Fanuc KAREL source: NC0015.KL

-- PROVISIONAL review KL for V940-1; original PC SHA256 a06a1c527e8287789b05f7df9faa5f540ba820ada4ca568a80dea30cb171e11d
-- Incomplete behavior may be omitted. Consult companion uncertainty JSON. Do not deploy.
PROGRAM NC0015
%NOLOCKGROUP
-- UNRESOLVED_LOCAL_POOL 1 cells at code offset 3; source declarations unknown
-- DIRECT_LOCAL_WORD_ACCESS alone does not prove INTEGER, REAL, or BOOLEAN
BEGIN
  -- V9_EXPOSED_INDEXED_TABLE_HINT layout=0001; 10 counted words exposed once; source arms/runtime held
  -- V9_CONDITION_STACK_HINT 5 bounded expression windows; static native code-base-relative target link; source arms held
  -- UNRESOLVED_PC offsets 0-8; opcodes 2B,2C,7B
  -- UNRESOLVED_PC offsets 13-20; opcodes 9D,23
  -- UNRESOLVED_PC offsets 25-38; opcodes 21,9D,57,79
  -- UNRESOLVED_PC offsets 43-61; opcodes 21,2E,52,23
  -- UNRESOLVED_PC offsets 66-71; opcodes 7A
  -- UNRESOLVED_PC offsets 76-89; opcodes 21,9D,57,79
  -- UNRESOLVED_PC offsets 94-112; opcodes 21,2E,52,23
  -- UNRESOLVED_PC offsets 117-122; opcodes 7A
  -- UNRESOLVED_PC offsets 127-140; opcodes 21,9D,57,79
  -- UNRESOLVED_PC offsets 145-163; opcodes 21,2E,52,23
  -- UNRESOLVED_PC offsets 168-173; opcodes 7A
  -- UNRESOLVED_PC offsets 178-191; opcodes 21,9D,57,79
  -- UNRESOLVED_PC offsets 196-214; opcodes 21,2E,52,23
  -- UNRESOLVED_PC offsets 219-224; opcodes 7A
  -- UNRESOLVED_PC offsets 229-242; opcodes 21,9D,57,79
  -- UNRESOLVED_PC offsets 247-265; opcodes 21,2E,52,23
  -- UNRESOLVED_PC offsets 270-275; opcodes 7A
  -- UNRESOLVED_PC offsets 280-294; opcodes 21,9D,52,23
  -- UNRESOLVED_PC offsets 324-328; opcodes 7F
  -- UNRESOLVED_PC offsets 333-337; opcodes 27,AA
  -- UNRESOLVED_PC offsets 342-346; opcodes 7F
END NC0015
